(*~
	<docu>
		<summary>
			Basic class for components.
		</summary>				
	</docu>	
~*)
FUNCTION_BLOCK ABSTRACT TcoComponent EXTENDS TcoObject IMPLEMENTS ITcoObject,ITcoRestorable, ITcoServiceable
VAR
	{attribute 'hide'}
	_serviceContexCycle : ULINT;	
(*~
	<docu>
		<summary>
			True if component is in service mode.
		</summary>			
	</docu>	
~*)
	{attribute addProperty Name "<#In service mode#>"}
	{attribute clr [ReadOnly()]}
	_inServiceMode : BOOL;	
END_VAR

CheckIfIsInServiceMode();

METHOD INTERNAL CheckIfIsInServiceMode 
VAR
	_myContextCycleCount : ULINT;
END_VAR
_myContextCycleCount := Context.StartCycleCount;
//When component.Service() is called "before" invoking its task _serviceContexCycle is equal to Context.StartCycleCount
//When component.Service() is called "after" invoking its task (_serviceContexCycle + 1) is equal to Context.StartCycleCount
//otherwise _serviceContexCycle should be lower then Context.StartCycleCount until Context.StartCycleCount overflow its range
//which should occur cca every 585 mil years at 1ms PLC task.    
_inServiceMode := _serviceContexCycle = _myContextCycleCount OR (_serviceContexCycle + 1) = _myContextCycleCount;
END_METHOD

METHOD FB_init : BOOL
VAR_INPUT
	bInitRetains : BOOL; // if TRUE, the retain variables are initialized (warm start / cold start)
	bInCopyCode : BOOL;  // if TRUE, the instance afterwards gets moved into the copy code (online change)
	Parent : ITcoObject;
END_VAR
SUPER^.FB_init(bInitRetains, bInCopyCode, Parent);
END_METHOD

(*~
	<docu>
		<summary>
			Gets whether the component is in serviceable state. Serviceable state is when ```Service``` method is called cyclicaly.   
		</summary>			
	</docu>	
~*)
PROPERTY IsService : BOOL
GET
CheckIfIsInServiceMode();
IsService := _inServiceMode;
END_GET
END_PROPERTY

(*~
	<docu>
		<summary>
			Restores this instance to the Ready state. Can be called explicitly or from within one of the restore mechanisms.	
		</summary>			
	</docu>	
~*)
METHOD ABSTRACT Restore : ITcoRestorable
END_METHOD

(*~
	<docu>
		<summary>
			Executes the logic for manual-maintenance control.   
		</summary>			
	</docu>	
~*)
METHOD PUBLIC FINAL Service
_serviceContexCycle := Context.StartCycleCount;
ServiceMode();
END_METHOD

(*~
	<docu>
		<summary>
		    Custom service (manual, maintenance) logic.
			This method must be implemented in derived class.
		</summary>			
	</docu>	
~*)
METHOD PROTECTED ABSTRACT ServiceMode
END_METHOD

END_FUNCTION_BLOCK

(* stored: Version 1.1.0.1, ProductVersion 3.1.4024.6
   POU TcoComponent: Id {8eb0512f-b833-4c04-bec5-9d60e2cb723b}, SpecialFunc None
   Method CheckIfIsInServiceMode: Id {f6d65f87-28bb-0f70-23ad-cefd8ddb093d}
   Method FB_init: Id {85de5686-5b6c-0496-3ce9-dba560b52906}
   Property IsService: Id {76fe61a9-82d7-035a-11e3-97101beac97d}
   Get Get: Id {c23442a0-b254-0ba9-01da-184a67a53561}
   Method Restore: Id {d0c02f91-fc49-4476-8612-b6c1e2ed01ac}
   Method Service: Id {c320b900-ed98-4dbe-a90b-28679bad227e}
   Method ServiceMode: Id {68a60f6a-9b62-45e9-a23f-6251b47fa211} *)
